Staubli VAL3: checkPoint.pgx

public program checkPoint(point x_PointToGo (dimensions=1), point x_PointStart (dimensions=1), bool& x_bUnreached[] (dimensions=1), tool x_tTool (dimensions=1), bool x_bLinear (dimensions=1))
  local joint jPoint
  local string message
  local num i
  local trsf t
begin
  // check if the point is null
  if (cycleStatus:bCycle==false and cycleStatus:bSimulation==false) or !x_bLinear
    x_bUnreached=false
    t=position(x_PointToGo,world)
    if t!={0,0,0,0,0,0}
      //
      // look if the point that you want to reach is valid
      if x_bLinear
        //
        // use the percentage....
        //
        for i=0.1 to 1 step 0.1
          pCheck.trsf=interpolateL(position(x_PointStart,world),position(x_PointToGo,world),i)
          x_bUnreached=!pointToJoint(x_tTool,herej(),pCheck,jPoint)
          if x_bUnreached
            return
          endIf
        endFor
      else
        // joint move or check only the working area
        x_PointToGo.config={sfree,efree,wfree}
        x_bUnreached=!pointToJoint(x_tTool,herej(),x_PointToGo,jPoint)
      endIf
    endIf
  endIf
end
